{attribute 'qualified_only'}
{attribute 'strict'}
{attribute 'to_string'}
TYPE E_MCS2OpMode :
(
    NONE := 0,
    // P-T-P target profil
    PROFILE_POSITION:=1,
    PROFIL_VELOCITY :=3,
    HOME:=6,
    // Cyclic synchronous modes
    CSP :=8,
    CSV :=9,
    CST := 10,
    CSTCA := 11,
    // smartAct MCS2 open loop
    CALIBRATE :=-1,
    STEP :=-4
) SINT;
END_TYPE

(* stored: Version 1.1.0.1
   DUT E_MCS2OpMode: Id {6b34f554-8c74-4ff3-b4ed-290b296a94b3} *)
